{attribute 'GeneratedUsingTerminal: AT2040-0250-0022'}
{attribute addProperty BoxType "AT2040-0250-0022"}
{attribute addProperty Id "A_0107_AT2000_5233_0018_AT2000_5233AT2000_33A3DF1B80"}
{attribute addProperty CRC "54382276"}
{attribute addProperty Size "80"}
TYPE A_0037_AT2040_0250_0022_033DCEC4 EXTENDS AT2040_A7FEA1CF :
STRUCT
	{attribute addProperty Name "A_0107_AT2000_5233_0018_AT2000_5233"}
	{attribute addProperty PreviousPort "A_0037(AT2040-0250-0022) : B"}
	A_0107_AT2000_5233_0018_AT2000_5233 : AT2000_33A3DF1B;
END_STRUCT
END_TYPE

(* stored: Version 1.2.0.0, ProductVersion 3.1.4024.9
   DUT A_0037_AT2040_0250_0022_033DCEC4: Id {132e9870-419b-4fb6-aaee-1d838d3de659} *)
